// TwinCAT 3 PLC project Test
// ProgramVersion: 3.1.0.8
// libraries:
//   FloatingPointUtils, * (System)
//   Tc2_ModbusSrv, * (Beckhoff Automation GmbH)
//   Tc2_Standard, * (Beckhoff Automation GmbH)
//   Tc2_System, * (Beckhoff Automation GmbH)
//   Tc2_Utilities, * (Beckhoff Automation GmbH)
//   Tc3_Interfaces, * (Beckhoff Automation GmbH)
//   Tc3_Module, * (Beckhoff Automation GmbH)
// project tree:
//   DUTs/ MODBUS_DATA_MAP.TcDUT
//   GVLs/ GVL.TcGVL
//   / PlcTask.TcTTO
//   POUs/ FB_CSV_Writer.TcPOU, FB_ModbusPoll.TcPOU, FB_ReadModbus.TcPOU, HexStringToReal.TcPOU, MAIN.TcPOU
// real-time tasks:
//   TASK PlcTask: cycle T#10ms, priority 20, ADS port 350

CONFIGURATION Test
    RESOURCE PLC ON TwinCAT3
        TASK PlcTask(INTERVAL := T#10ms, PRIORITY := 20);
        PROGRAM MAIN WITH PlcTask : MAIN;
    END_RESOURCE
END_CONFIGURATION

// ---- DUTs/MODBUS_DATA_MAP.TcDUT
TYPE MODBUS_DATA_MAP :
STRUCT
	_ipAddress : STRING;
	_startAddress : WORD;
END_STRUCT
END_TYPE

// ---- GVLs/GVL.TcGVL
VAR_GLOBAL
END_VAR

// ---- POUs/MAIN.TcPOU
PROGRAM MAIN 
VAR

fbReadmb : FB_ReadModbus ;
arr: ARRAY [0..1] OF MODBUS_DATA_MAP;
data : ARRAY[0..1] OF REAL;
END_VAR

arr[0]._ipAddress := '192.168.1.101';
arr[1]._ipAddress := '192.168.1.101';
arr[0]._startAddress := 0;
arr[1]._startAddress := 12;

fbReadmb(inputData := arr , dataArr => data);

END_PROGRAM

// ---- POUs/FB_ReadModbus.TcPOU
FUNCTION_BLOCK FB_ReadModbus
VAR_INPUT
inputData : ARRAY[0..1] OF MODBUS_DATA_MAP;
intervalToSampleData : TIME := T#5S; //modbus update rate (lower rate = more disk usage) default : 5 seconds
fileName: STRING := 'data';//changinng this will change the file otherwise it will overwrite the data : default 'data'
END_VAR
VAR_OUTPUT
	dataArr : ARRAY[0..1] OF REAL;
END_VAR
VAR
	
mb1 : FB_ModbusPoll; //first poller
mb2 : FB_ModbusPoll; // second  poller

bex : BOOL; //delay bit
rex : BOOL;	//other delay bit

dataWriter : FB_CSV_Writer; //fb that writes data to a csv file 

timer  : TON; //timer to coordinate when to write to the file (basically the update rate of the modbus server)

exBit : BOOL := TRUE; //excute bit for the timer

numberOfReadingsTaken : INT;//holds how many readings have been taken from initial download

END_VAR

mb1.ipAd := inputData[0]._ipAddress;
mb1.startAddr := inputData[0]._startAddress;
mb2.ipAd := inputData[1]._ipAddress;
mb2.startAddr := inputData[1]._startAddress;


//5 second timeout
timer.PT := intervalToSampleData;

IF bex THEN
	mb1(value => dataArr[0]);
ELSE
	mb2(value => dataArr[1]);
END_IF

//some bit delays
IF NOT bex THEN
	bex := NOT bex;
ELSE 
	bex := rex;
END_IF

rex := NOT rex;

//timer starts when execute bit is true
timer(in:= exBit);

//if it is running write false
IF NOT timer.Q THEN
	//start timer
	exBit := TRUE;
	//falseify the write line	
	dataWriter(bWriteLine := FALSE, sFileName := fileName , fDataPoint1 := dataArr[0] , fDataPoint2 := dataArr[1]);
ELSE	
	//reset the bit to reset the timer
	exBit := FALSE;	
	//write the data
	dataWriter(bWriteLine := TRUE, sFileName := fileName , fDataPoint1 := dataArr[0] , fDataPoint2 := dataArr[1]);
	//bump up the readings
	numberOfReadingsTaken:=numberOfReadingsTaken+1;
END_IF

END_FUNCTION_BLOCK

// ---- POUs/FB_ModbusPoll.TcPOU
FUNCTION_BLOCK FB_ModbusPoll

VAR_INPUT
	ipAd : STRING; // the ip address of the modbus server
	startAddr : WORD; // the start address
END_VAR

VAR_OUTPUT
	value : REAL;
END_VAR

VAR
	dataStr :STRING;
	bModbusTick : BOOL;
	fbReadRegs : FB_MBReadInputRegs;
	converter : HexStringToReal;
	arr : ARRAY [0..2] OF WORD;
END_VAR


//setup the modbus block
fbReadRegs.sIPAddr := ipAd; //gateway ip
fbReadRegs.nTCPPort := MODBUS_TCP_PORT; //502
fbReadRegs.nUnitID := 16#FF; //255
fbReadRegs.nQuantity := 3; //3 words
fbReadRegs.tTimeout := T#5S; //30 sec timout
fbReadRegs.nMBAddr := startAddr;
fbReadRegs.cbLength := 6;//nq*2
fbReadRegs.pDestAddr := ADR(arr); //the pointer to the array

//the rising edge of the input negate the tick to create  a rising input of change :)
fbReadRegs.bExecute := (bModbusTick := NOT bModbusTick); 

//uppercase(convert first number to hex + convert second number to hex)
dataStr := F_TOUCase(CONCAT(WORD_TO_HEXSTR(arr[1],4,TRUE),WORD_TO_HEXSTR(arr[2],4,TRUE))); 
fbReadRegs();

//use converter to convert last 2 words to a fp value
converter(str:=dataStr, out => value);

END_FUNCTION_BLOCK

// ---- POUs/HexStringToReal.TcPOU
FUNCTION_BLOCK HexStringToReal
VAR_INPUT
	str :STRING;
END_VAR
VAR_OUTPUT
	out : REAL;
END_VAR
VAR
holdStr : STRING := '';
binStr : STRING := '';
bin : STRING := '';	
sExponent : INT := 1;
expVal : INT;
sMantissa : STRING;
i :INT :=0;
ar : ARRAY[0..23] OF STRING;

significand : REAL;
decVal : REAL ;
END_VAR

FOR i :=1 TO 8 BY 1 DO
	holdStr := MID(str,1,i);
	
	IF holdStr = '0' THEN
		bin := '0000';
	ELSIF holdStr = '1' THEN
		bin := '0001';
	ELSIF holdStr = '2' THEN
		bin := '0010';
	ELSIF holdStr = '3' THEN
		bin := '0011';
	ELSIF holdStr = '4' THEN
		bin := '0100';
	ELSIF holdStr = '5' THEN
		bin := '0101';
	ELSIF holdStr = '6' THEN
		bin := '0110';
	ELSIF holdStr = '7' THEN
		bin := '0111';
	ELSIF holdStr = '8' THEN
		bin := '1000';
	ELSIF holdStr = '9' THEN
		bin := '1001';
	ELSIF holdStr = 'A' THEN
		bin := '1010';
	ELSIF holdStr = 'B' THEN
		bin := '1011';
	ELSIF holdStr = 'C' THEN
		bin := '1100';
	ELSIF holdStr = 'D' THEN
		bin := '1101';
	ELSIF holdStr = 'E' THEN
		bin := '1110';
	ELSIF holdStr = 'F' THEN
		bin := '1111';
	END_IF
	
	binStr := CONCAT(binStr,bin);
		
END_FOR

binStr := RIGHT(binStr,32);
binStr := DELETE(binStr,1,1);

sExponent := STRING_TO_INT(CONCAT('2#',LEFT(binStr,8))) - 127;
sMantissa := MID(binStr,23,9);

decVal := 0.5;
significand := 0;

FOR i := 0 TO 23 BY 1 DO
	ar[i] := MID(sMantissa,1,i);
END_FOR

FOR i:= 1 TO 23 BY 1 DO
	significand := significand + (STRING_TO_INT(ar[i])*decVal);
	decVal := decVal/2;
END_FOR

expVal := 2;
FOR i:= 0 TO sExponent-2 BY 1 DO
	expVal := 2*expVal;
END_FOR

out := (significand +1) * (expVal);
RETURN;

END_FUNCTION_BLOCK

// ---- POUs/FB_CSV_Writer.TcPOU
FUNCTION_BLOCK FB_CSV_Writer //Matt
VAR_INPUT
	bWriteLine:	BOOL; //true if you want to write to the file
	sFileName:	STRING; //name of the file to write
	fDataPoint1:	REAL; //data point 1
	fDataPoint2:	REAL; //data point 2
END_VAR
VAR_OUTPUT
	bBusy:	BOOL;
	bError:	BOOL;
	sError:	STRING;
END_VAR
VAR
	fbFileOpen:	FB_FileOpen; //fb to open the file to begin appending
	fbFilePuts:	FB_FilePuts; //fb to write to the file
	fbFileClose: FB_FileClose; // closes the file
	
	rtWrite:	R_TRIG; //trigger
	
	fbGetSystemTime : GETSYSTEMTIME;
	fileTime : T_FILETIME;
	
	nState:	INT; //state to cycle to parts of appending
	sTempPathName:	STRING; 
	sDataString:	STRING; //string to write
END_VAR

rtWrite(CLK := bWriteLine);

CASE nState OF
	0:	(*IDLE*)
		bBusy := FALSE;
		IF rtWrite.Q THEN
			sTempPathName := CONCAT(CONCAT('C:\Temp\',sFileName),'.csv');
			fbGetSystemTime(timeLoDW=>fileTime.dwLowDateTime, timeHiDW=>fileTime.dwHighDateTime );
			sDataString := CONCAT(CONCAT(CONCAT( CONCAT(CONCAT(REAL_TO_STRING(fDataPoint1),',') ,REAL_TO_STRING(fDataPoint2)),','),SYSTEMTIME_TO_STRING( FILETIME_TO_SYSTEMTIME( fileTime ) ) ),'$N'); 
			bBusy := TRUE;
			bError := FALSE;
			sError := '';
			nState := nState + 10;
		END_IF		
	
	10:	(*Open File*)	
		fbFileOpen(	sPathName := sTempPathName,nMode := FOPEN_MODEAPPEND,bExecute := TRUE,tTimeOut := T#1S);
		IF NOT fbFileOpen.bBusy THEN
			fbFileOpen(	bExecute := FALSE);
			IF fbFileOpen.bError THEN
				bError := TRUE;
				sError := 'Could Not Open File';
				nState := 0;
			ELSE
				nState := nState + 10;
			END_IF
		END_IF
		
	20:	(*Write Line To File*)
		fbFilePuts(	hFile := fbFileOpen.hFile,sLine := sDataString,bExecute := TRUE,tTimeout := T#1S);
		IF NOT fbFilePuts.bBusy THEN
			fbFilePuts(	bExecute := FALSE);
			IF fbFilePuts.bError THEN
				bError := TRUE;
				sError := 'Could not write to file';
				nState := nState + 10;
			ELSE
				nState := nState + 10;
			END_IF
		END_IF
		
	30:	(*Close File*)
		fbFileClose(hFile := fbFileOpen.hFile,bExecute := TRUE,tTimeout := T#1S);
		IF NOT fbFileClose.bBusy THEN
			fbFileClose(	bExecute := FALSE);
			IF fbFileClose.bError THEN
				bError := TRUE;
				sError := 'Could not close file';
				nState := 0;
			ELSE
				nState := 0;
			END_IF
		END_IF
END_CASE

END_FUNCTION_BLOCK
